FUNCTION_BLOCK E_PERMIT (* Permissive propagation of an event *)
  (* Standard: 61499-1-A.1 *)
  (* Version 0.2, 2012-12-20, IH, TU Wien, added service sequences for test case specification *)
  (* Version 0.1, 2003-12-30, JHC, Rockwell Automation, Updated for 61499-1 CDV. *)
  (* Version 0.0, 2001-03-03, JHC, Rockwell Automation *)
  (* Compiler header: package fb.rt.events; *)
  (* Compiler Java IBM VisualAge 3.0 *)
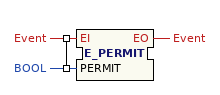
  EVENT_INPUT
    EI WITH PERMIT; (* Event input *)
  END_EVENT
  EVENT_OUTPUT
    EO; (* Event output *)
  END_EVENT
  VAR_INPUT
    PERMIT : BOOL;
  END_VAR
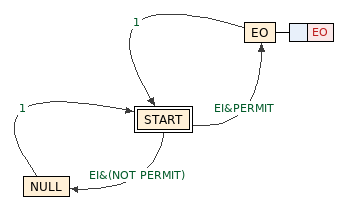
  EC_STATES
    START; (* Initial State *)
    EO : -> EO; (* Issue EO Event *)
    NULL; (* Do nothing if PERMIT=FALSE *)
  END_STATES
  EC_TRANSITIONS
    START TO EO := EI&PERMIT;
    EO TO START := 1;
    START TO NULL := EI&(NOT PERMIT);
    NULL TO START := 1;
  END_TRANSITIONS
  SERVICE FB Interface/Runtime Environment (* Permissive propagation of an event *)
    SEQUENCE EventTerminationTest
      FB Interface.EI(PERMIT:=FALSE;);
    END_SEQUENCE
    SEQUENCE EventPropagationTest
      FB Interface.EI(PERMIT:=TRUE;) -> FB Interface.EO();
    END_SEQUENCE
    SEQUENCE Negative Test
      FB Interface.EI(PERMIT:=true;);
    END_SEQUENCE
  END_SERVICE
END_FUNCTION_BLOCK
